// TIA Portal V20 export
DATA_BLOCK "ReportValues_DB"   // DB35
AUTHOR : Siemens AG
FAMILY : ServiceControl
VERSION : 1.0
// stored: InstanceOfName ReportValues, InstanceOfType FB
"ReportValues"
   // VAR
   //    MTPAnalog { S7_SetPoint := 'True'} : Array[0..10] of "UDT_MTP_AnaReportValue";
   //    MTPDigital { S7_SetPoint := 'True'} : Array[0..0] of "UDT_MTP_DIntReportValue";
   //    MTPBinary { S7_SetPoint := 'True'} : Array[0..2] of "UDT_MTP_BinReportValue";
   //    MTPString { S7_SetPoint := 'True'} : Array[0..0] of "UDT_MTP_StringReportValue";
   // END_VAR
BEGIN
   MTPAnalog[0..9].V := 0.0;
   MTPAnalog[0..9].VSclMin := 0.0;
   MTPAnalog[0..1].VSclMax := 3000.0;
   MTPAnalog[2..3].VSclMax := 100.0;
   MTPAnalog[4..5].VSclMax := 3000.0;
   MTPAnalog[6..7].VSclMax := 100.0;
   MTPAnalog[8].VSclMax := 3000.0;
   MTPAnalog[9].VSclMax := 1.0;
   MTPAnalog[0..1].VUnit := 1038;
   MTPAnalog[2..3].VUnit := 1001;
   MTPAnalog[4..5].VUnit := 1038;
   MTPAnalog[6..7].VUnit := 1001;
   MTPAnalog[8].VUnit := 1038;
   MTPAnalog[9].VUnit := 1000;
   MTPBinary[0..1].V := False;
   MTPBinary[0..1].VState0 := '';
   MTPBinary[0..1].VState1 := '';
END_DATA_BLOCK
